Omron CX-Programmer project NewProject (CX-Programmer 9.75)

# PLC CIRCUIT_DISTRIBUTING_PATCH_1: CP2E-N N

## Global symbols (name address type ; comment)
0.00 BOOL  ; B-ON
0.01 BOOL  ; B-OFF
0.05 BOOL  ; S-SL-MAJU
0.06 BOOL  ; S-AR-KIRI
0.07 BOOL  ; S-AR-KANAN
0.08 BOOL  ; S-BENDA-KIRI
0.09 BOOL  ; S-VACCUM
0.10 BOOL  ; S-BENDA-KANAN
100.00 BOOL  ; SL-MAJU
100.01 BOOL  ; AR-KANAN
100.02 BOOL  ; AR-KIRI
100.03 BOOL  ; VACCUM
100.04 BOOL  ; BLOW
200.00 BOOL  ; K-UTAMA
200.08 BOOL  ; K-LOOP

## Program NewProgram1 (cyclic task 0)
; SDS

### Section Section1
; SDS
; rung 0: # CIRCUIT DISTRIBUTING PACTH 1 / JOBSHEET MEKATRONIKA 2025/2026 / DATE : 21/07/2025 / BY     : CALYA KIEZA ATAFADILA (XII TM A) / VARIABLES / - K   = KONTAKTOR / - L    = LAMPU / - AR  = ARM (LENGAN) / - B    = BUTTON / - S    = SENSOR / - SL  = SILINDER
; rung 1: SYSTEM

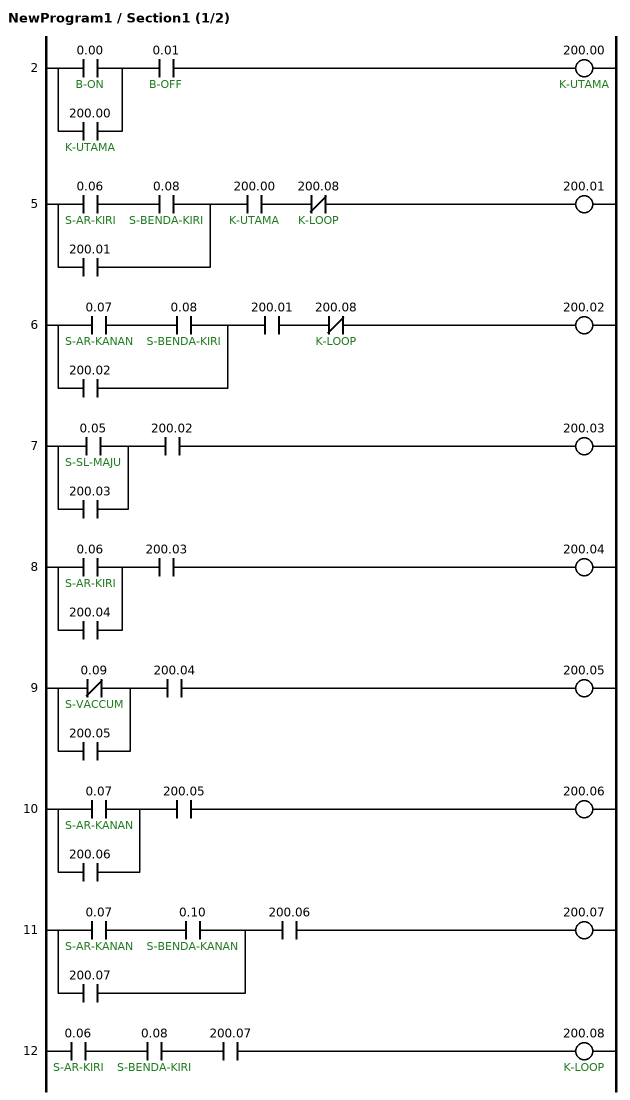
; rung 2
LD 0.00  ; B-ON
OR 200.00  ; K-UTAMA
AND 0.01  ; B-OFF
OUT 200.00  ; K-UTAMA
; rung 4: CONTROL
; rung 5
LD 0.06  ; S-AR-KIRI
AND 0.08  ; S-BENDA-KIRI
OR 200.01
AND 200.00  ; K-UTAMA
ANDNOT 200.08  ; K-LOOP
OUT 200.01
; rung 6
LD 0.07  ; S-AR-KANAN
AND 0.08  ; S-BENDA-KIRI
OR 200.02
AND 200.01
ANDNOT 200.08  ; K-LOOP
OUT 200.02
; rung 7
LD 0.05  ; S-SL-MAJU
OR 200.03
AND 200.02
OUT 200.03
; rung 8
LD 0.06  ; S-AR-KIRI
OR 200.04
AND 200.03
OUT 200.04
; rung 9
LDNOT 0.09  ; S-VACCUM
OR 200.05
AND 200.04
OUT 200.05
; rung 10
LD 0.07  ; S-AR-KANAN
OR 200.06
AND 200.05
OUT 200.06
; rung 11
LD 0.07  ; S-AR-KANAN
AND 0.10  ; S-BENDA-KANAN
OR 200.07
AND 200.06
OUT 200.07
; rung 12
LD 0.06  ; S-AR-KIRI
AND 0.08  ; S-BENDA-KIRI
AND 200.07
OUT 200.08  ; K-LOOP
; rung 14: LAMP

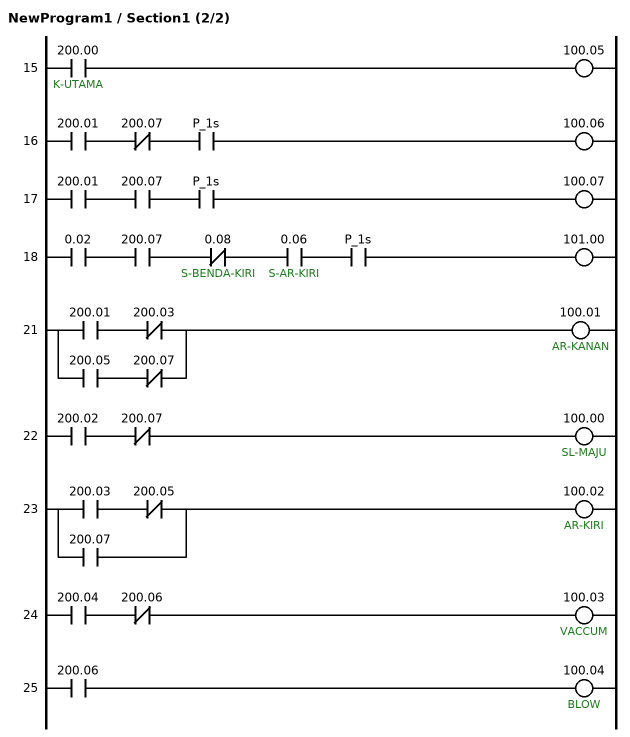
; rung 15
LD 200.00  ; K-UTAMA
OUT 100.05
; rung 16
LD 200.01
ANDNOT 200.07
AND P_1s
OUT 100.06
; rung 17
LD 200.01
AND 200.07
AND P_1s
OUT 100.07
; rung 18
LD 0.02
AND 200.07
ANDNOT 0.08  ; S-BENDA-KIRI
AND 0.06  ; S-AR-KIRI
AND P_1s
OUT 101.00
; rung 20: OUTPUT
; rung 21
LD 200.01
ANDNOT 200.03
LD 200.05
ANDNOT 200.07
ORLD
OUT 100.01  ; AR-KANAN
; rung 22
LD 200.02
ANDNOT 200.07
OUT 100.00  ; SL-MAJU
; rung 23
LD 200.03
ANDNOT 200.05
OR 200.07
OUT 100.02  ; AR-KIRI
; rung 24
LD 200.04
ANDNOT 200.06
OUT 100.03  ; VACCUM
; rung 25
LD 200.06
OUT 100.04  ; BLOW

### Section END
; rung 0
END(001)